ABB RobotStudio station: zaliczenie_zadanie1_20200111-225542.rsstn

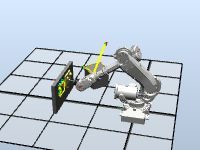
Station zaliczenie_zadanie1 (saved by RobotStudio 6.8.8307.1040)
Controller IRB_6640_185kg_2.80m
  mechanical unit ROB_1: IRB6640_185_280__04, 6 joints, base frame (0, 0, 0) mm
Layout (positions relative to the parent item):
  - IRB6640_185_280__04 [mechanism, from Robots\IRB6640_185_280_G_04.rslib] at (0, 0, 0) mm; joint values [-1.4668, -0.6795, -3.0641, 0.1316, 0.8694, 3.0294] (rad or m)
  - Part_13 [part]
  - Part_14 [part] at (132.45, 1287.69, 0) mm
  - Part_20 [part] at (0, 0, 10) mm
  - Part_21 [part] at (0, 0, 10) mm
  - Part_34 [part]
  - dupsko_bonczura [mechanism] at (-144.3, 1575.65, 714.65) mm, rotated rx 0 ry 75 rz 90 deg
      TCP dupsko_bonczura at (65.7, 0, 297.48) mm, rotated rx 0 ry 15 rz 0 deg
      links: Part_42
  - Part_48 [part]
  - Part_58 [part]
  - Part_59 [part] at (391.01, 977.32, 0) mm
  - Part_60 [part] at (1091.01, 977.32, 0) mm, rotated rx 0 ry 0 rz 45 deg
  - Part_61 [part] at (1091.01, 977.32, 0) mm, rotated rx 0 ry 0 rz 45 deg
  - Part_70 [part] at (-116.27, 0, -471.82) mm
Attachment: dupsko_bonczura is attached to IRB6640_185_280__04 / Link6
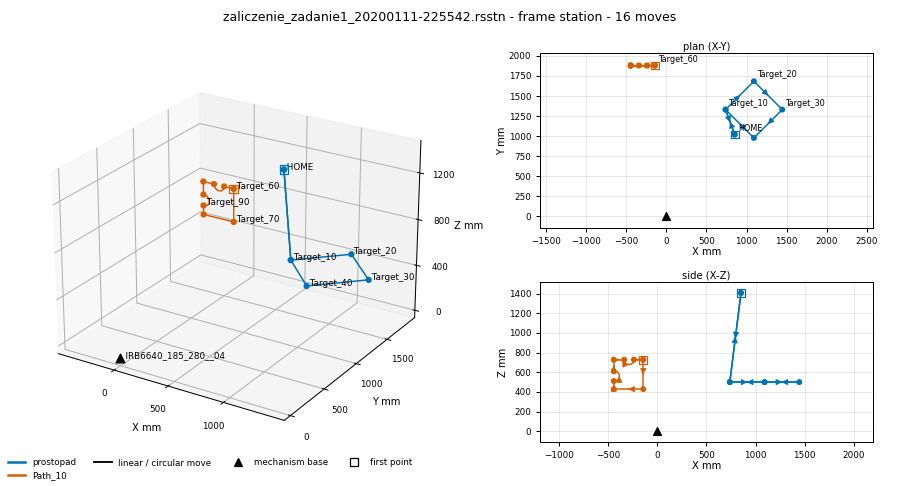
[picture p0: tool path of zaliczenie_zadanie1_20200111-225542.rsstn in frame station, 16 of 16 moves have a stored position in this frame; points joined in program order, loops and branches not executed]
Targets, tools, work objects and paths stored in the station, written as RAPID:
! task T_ROB1
MODULE CalibData
  PERS tooldata MyNewTool:=[TRUE,[[489.305,-400.511,237.057],[0.965925826,0,0.258819045,0]],[1,[0,0,1],[1,0,0,0],0,0,0]];
  PERS tooldata dupsko_bonczura:=[TRUE,[[65.705,0,297.481],[0.991444861,0,0.130526192,0]],[1,[0,0,1],[1,0,0,0],0,0,0]];
ENDMODULE

! task T_ROB1
MODULE Module1
  CONST robtarget HOME:=[[851.118384663,1020.171891437,1407.621949555],[0.030067928,-0.678210327,0.729882518,-0.079988635],[-2,1,-1,6],[9E+09,9E+09,9E+09,9E+09,9E+09,9E+09]];
  CONST robtarget Target_10:=[[737.455573018,1330.871650409,500],[0,-0.382683432,0.923879533,0],[-2,1,0,6],[9E+09,9E+09,9E+09,9E+09,9E+09,9E+09]];
  CONST robtarget Target_20:=[[1091.008963611,1684.425041002,500],[0,-0.382683432,0.923879533,0],[-2,1,0,6],[9E+09,9E+09,9E+09,9E+09,9E+09,9E+09]];
  CONST robtarget Target_30:=[[1444.562354205,1330.871650409,500],[0,-0.382683432,0.923879533,0],[-2,0,1,7],[9E+09,9E+09,9E+09,9E+09,9E+09,9E+09]];
  CONST robtarget Target_40:=[[1091.008963611,977.318259815,500],[0,-0.382683432,0.923879533,0],[-2,0,1,7],[9E+09,9E+09,9E+09,9E+09,9E+09,9E+09]];
  CONST robtarget Target_50:=[[737.455573018,1330.871650409,500],[0,-0.382683432,0.923879533,0],[-2,-1,-2,7],[9E+09,9E+09,9E+09,9E+09,9E+09,9E+09]];
  CONST robtarget Target_60:=[[-144.296598994,1880,728.176467536],[0.5,-0.5,0.5,0.5],[-1,0,1,6],[9E+09,9E+09,9E+09,9E+09,9E+09,9E+09]];
  CONST robtarget Target_70:=[[-144.296598994,1880,428.176467536],[0.5,-0.5,0.5,0.5],[-1,0,1,6],[9E+09,9E+09,9E+09,9E+09,9E+09,9E+09]];
  CONST robtarget Target_80:=[[-444.296598994,1880,428.176467536],[0.5,-0.5,0.5,0.5],[-1,0,1,6],[9E+09,9E+09,9E+09,9E+09,9E+09,9E+09]];
  CONST robtarget Target_90:=[[-444.296598994,1880,510.750512977],[0.5,-0.5,0.5,0.5],[-1,0,1,6],[9E+09,9E+09,9E+09,9E+09,9E+09,9E+09]];
  CONST robtarget Target_100:=[[-386.8491628,1880,560.192759023],[0.5,-0.5,0.5,0.5],[-1,0,1,6],[9E+09,9E+09,9E+09,9E+09,9E+09,9E+09]];
  CONST robtarget Target_110:=[[-444.296598994,1880,609.63500507],[0.5,-0.5,0.5,0.5],[-1,0,1,6],[9E+09,9E+09,9E+09,9E+09,9E+09,9E+09]];
  CONST robtarget Target_120:=[[-444.296598994,1880,728.176467536],[0.5,-0.5,0.5,0.5],[-1,0,1,6],[9E+09,9E+09,9E+09,9E+09,9E+09,9E+09]];
  CONST robtarget Target_130:=[[-338.609598994,1880,728.176467536],[0.5,-0.5,0.5,0.5],[-1,0,1,6],[9E+09,9E+09,9E+09,9E+09,9E+09,9E+09]];
  CONST robtarget Target_140:=[[-288.609598994,1880,678.176467536],[0.5,-0.5,0.5,0.5],[-1,0,1,6],[9E+09,9E+09,9E+09,9E+09,9E+09,9E+09]];
  CONST robtarget Target_150:=[[-238.609598994,1880,728.176467536],[0.5,-0.5,0.5,0.5],[-1,0,1,6],[9E+09,9E+09,9E+09,9E+09,9E+09,9E+09]];
  CONST robtarget Target_160:=[[-144.296598994,1880,728.176467536],[0.5,-0.5,0.5,0.5],[-1,0,1,6],[9E+09,9E+09,9E+09,9E+09,9E+09,9E+09]];
  PROC prostopad()
    MoveL HOME,vmax,z100,dupsko_bonczura\WObj:=wobj0;
    MoveL Target_10,v1000,fine,dupsko_bonczura\WObj:=wobj0;
    MoveL Target_20,v100,fine,dupsko_bonczura\WObj:=wobj0;
    MoveL Target_30,v100,fine,dupsko_bonczura\WObj:=wobj0;
    MoveL Target_40,v100,fine,dupsko_bonczura\WObj:=wobj0;
    MoveL Target_50,v100,fine,dupsko_bonczura\WObj:=wobj0;
    MoveL HOME,v1000,z100,dupsko_bonczura\WObj:=wobj0;
  ENDPROC
  PROC Path_10()
    MoveL Target_60,v1000,fine,dupsko_bonczura\WObj:=wobj0;
    MoveL Target_70,v100,fine,dupsko_bonczura\WObj:=wobj0;
    MoveL Target_80,v100,fine,dupsko_bonczura\WObj:=wobj0;
    MoveL Target_90,v100,fine,dupsko_bonczura\WObj:=wobj0;
    MoveC Target_100,Target_110,v100,fine,dupsko_bonczura\WObj:=wobj0;
    MoveL Target_120,v100,fine,dupsko_bonczura\WObj:=wobj0;
    MoveL Target_130,v100,fine,dupsko_bonczura\WObj:=wobj0;
    MoveC Target_140,Target_150,v100,fine,dupsko_bonczura\WObj:=wobj0;
    MoveL Target_160,v100,fine,dupsko_bonczura\WObj:=wobj0;
  ENDPROC
ENDMODULE

